FUNCTION_BLOCK Test_NotificationNoArgs EXTENDS tcl_SimpleUnitTestLibrary.T_UnitTestBase
VAR
    Source   : T_Notification;
    Handler  : T_NotificationHandler;
    IsRaised : BOOL;
END_VAR

Handler.FB_init(bInitRetains := FALSE,
                bInCopyCode  := FALSE);

Source.ClearNotificationHandlers().AddNotificationHandler(Handler);

Source.Raise();
IsRaised := Handler.IsRaised();

Assertion.AssertEquals_BOOL(Expected     := TRUE,
                            Actual       := IsRaised,
                            VariableName := 'IsRaised');

TestFinished();

END_FUNCTION_BLOCK

(* stored: Version 1.1.0.1, ProductVersion 3.1.4024.9
   POU Test_NotificationNoArgs: Id {cc5ef7a4-9804-419b-b45f-a2befe39c1e5}, SpecialFunc None *)
